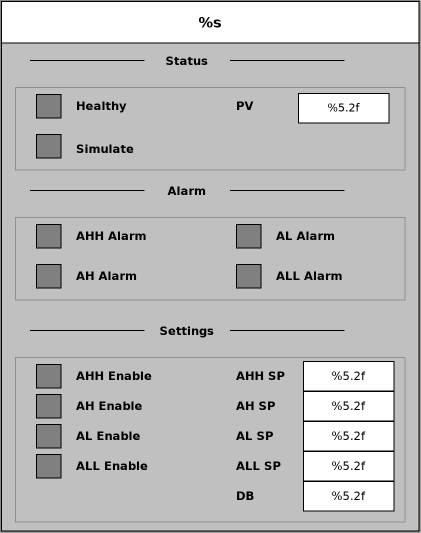
VISUALIZATION AIN_Template  // 421x533
VAR_IN_OUT
	DUT								: DUT_AIN;
END_VAR
    Group (1,1 418x530)
        Rectangle (0,0 418x530)
        Rectangle (0,0 418x42)
    Textfield (1,4 418x37), "%s", text variable: DUT.AIN_ID
    Line (30,330) (144,330)
    Line (230,330) (344,330)
    GroupBox (15,349 390x173)
        RoundedRectangle (21,45 25x24), colour toggle: DUT.AH_Enable
            toggle DUT.AH_Enable
        RoundedRectangle (21,75 25x24), colour toggle: DUT.AL_Enable
            toggle DUT.AL_Enable
        RoundedRectangle (21,105 25x24), colour toggle: DUT.ALL_Enable
            toggle DUT.ALL_Enable
        Label (218,42 64x30), "AH SP"
        Label (218,72 64x30), "AL SP"
        Label (218,102 64x30), "ALL SP"
        Label (218,132 64x30), "DB"
    RoundedRectangle (36,364 25x24), colour toggle: DUT.AHH_Enable
        toggle DUT.AHH_Enable
    Label (73,361 100x30), "AHH Enable"
    Label (233,361 64x30), "AHH SP"
    Label (112,316 150x30), "Settings"
    Label (73,391 100x30), "AH Enable"
    Label (73,421 100x30), "AL Enable"
    Label (73,451 100x30), "ALL Enable"
    Rectangle (303,361 91x30), "%5.2f", text variable: DUT.AHH_SP
        OnMouseClick: write DUT.AHH_SP via Default
    Rectangle (303,391 91x30), "%5.2f", text variable: DUT.AH_SP
        OnMouseClick: write DUT.AH_SP via Default
    Rectangle (303,421 91x30), "%5.2f", text variable: DUT.AL_SP
        OnMouseClick: write DUT.AL_SP via Default
    Rectangle (303,451 91x30), "%5.2f", text variable: DUT.ALL_SP
        OnMouseClick: write DUT.ALL_SP via Default
    Rectangle (303,481 91x30), "%5.2f", text variable: DUT.DB
        OnMouseClick: write DUT.DB via Default
    Line (30,60) (144,60)
    Line (230,60) (344,60)
    GroupBox (15,79 390x91)
        Label (218,12 64x30), "PV"
        Rectangle (283,14 91x30), "%5.2f", text variable: DUT.PV
            OnMouseClick: write DUT.PV via Default
    RoundedRectangle (36,94 25x24), colour toggle: DUT.Healthy
    Label (73,91 64x30), "Healthy"
    Label (73,134 64x30), "Simulate"
    RoundedRectangle (36,134 25x24), colour toggle: DUT.Simulate
        toggle DUT.Simulate
    Label (112,46 150x30), "Status"
    Line (30,190) (144,190)
    Line (230,190) (344,190)
    GroupBox (15,209 390x91)
        RoundedRectangle (21,55 25x24), colour toggle: DUT.AH
        RoundedRectangle (221,55 25x24), colour toggle: DUT.ALL
    RoundedRectangle (36,224 25x24), colour toggle: DUT.AHH
    Label (73,221 100x30), "AHH Alarm"
    Label (112,176 150x30), "Alarm"
    Label (73,261 100x30), "AH Alarm"
    RoundedRectangle (236,224 25x24), colour toggle: DUT.AL
    Label (273,221 100x30), "AL Alarm"
    Label (273,261 100x30), "ALL Alarm"
END_VISUALIZATION

(* stored: Version 1.1.0.1, ProductVersion 3.1.4022.18
   Visu AIN_Template: Id {8ec24bbe-a78d-4f7c-8dcb-c4c1bb08b452} *)
